{attribute 'linkalways'} 
{attribute 'no_explicit_call' := 'This FB is a CLASS and must be accessed using methods or properties'}
{attribute 'enable_dynamic_creation'}
FUNCTION_BLOCK ChunkedResponseData EXTENDS Disposable IMPLEMENTS I_ChunkedResponseData
VAR
	pData : POINTER TO BYTE;
	size : UDINT;
	currentPointerLocation : PVOID;
	remainingLengthToSendInBytes : UDINT;
END_VAR

METHOD FB_exit : BOOL
VAR_INPUT
	bInCopyCode : BOOL; // if TRUE, the exit method is called for exiting an instance that is copied afterwards (online change).
END_VAR
IF bInCopyCode THEN
	RETURN;
END_IF

IF pData <> 0 THEN
	__DELETE(pData);
END_IF
END_METHOD

METHOD FB_init : BOOL
VAR_INPUT
	bInitRetains : BOOL; // if TRUE, the retain variables are initialized (warm start / cold start)
	bInCopyCode : BOOL;  // if TRUE, the instance afterwards gets moved into the copy code (online change)
	Address : PVOID;
	Size : UDINT;
END_VAR
StoreData(Address, Size);
END_METHOD

PROPERTY PUBLIC SendComplete : BOOL
GET
SendComplete := remainingLengthToSendInBytes = 0;
END_GET
END_PROPERTY

METHOD PUBLIC SendNextChunk
VAR_INPUT
	Response : I_ServerResponse;
	Size : UDINT;
END_VAR
VAR
	sendSize : UDINT;
END_VAR
IF SendComplete THEN 
	Response.Error('BAD_REQUEST', 'No further data to send');
	RETURN;
END_IF

sendSize := Size - 1;

IF Size > remainingLengthToSendInBytes THEN 
	sendSize := remainingLengthToSendInBytes;
END_IF

Response.SuccessWithPayload(currentPointerLocation, sendSize);

currentPointerLocation := currentPointerLocation + sendSize;
remainingLengthToSendInBytes := remainingLengthToSendInBytes - sendSize;
END_METHOD

PROPERTY SizeRemaining : UDINT
GET
SizeRemaining := remainingLengthToSendInBytes;
END_GET
END_PROPERTY

METHOD PRIVATE StoreData
VAR_INPUT
	Address : PVOID;
	Size : UDINT;
END_VAR
pData := __NEW(BYTE, Size);
THIS^.size := Size;
memcpy(pData, Address, Size);
currentPointerLocation := pData;
remainingLengthToSendInBytes := Size;
END_METHOD

END_FUNCTION_BLOCK

(* stored: Version 1.1.0.1, ProductVersion 3.1.4026.13
   POU ChunkedResponseData: Id {781f9fc5-3ebc-4ff0-ac98-856e05f50372}, SpecialFunc None
   Folder Constructor: Id {c80cbdb3-cb9a-49fe-9914-91d60f1c0ad0}
   Folder Destructor: Id {c8a95ce9-85c1-4947-8c24-4259ab62db6f}
   Folder Private: Id {aa8b3d89-0333-425f-8039-0af43cf40e23}
   Method FB_exit: Id {26a59a06-9389-4457-b5a3-0891228185bf}
   Method FB_init: Id {c8bcd570-a5c0-402b-9d22-4c3fe10c9f06}
   Property SendComplete: Id {0e3ef159-392b-4b06-885d-1d84746037be}
   Get Get: Id {2193082c-2fb6-4f72-a650-476ec7e26479}
   Method SendNextChunk: Id {6566f4d7-cb0d-4093-a982-79ab5b2f23da}
   Property SizeRemaining: Id {da39f145-753d-4410-ba23-30977ba1ac28}
   Get Get: Id {52c6e58e-8432-4843-ba02-503e5f766076}
   Method StoreData: Id {05fe66e7-cab7-4f49-a1e8-1358584c2b63} *)
